(* IEC 61131-3 sources: RL_MAR/experiments/comparison/autoplc/results/deepseek-ai-DeepSeek-V3.2_20260508_111905/hard_92, 1 file *)

(* ---- hard_92_1.st ---- *)
FUNCTION_BLOCK FB_BreakerControlSystem
VAR_INPUT
    B10_1_Trip : BOOL;
    B10_1_Close : BOOL;
    B10_2_Trip : BOOL;
    B10_2_Close : BOOL;
    B10_12_Trip : BOOL;
    B10_12_Close : BOOL;
    B54_Trip : BOOL;
    B54_Close : BOOL;
    B55_Trip : BOOL;
    B55_Close : BOOL;
    B56_Trip : BOOL;
    B56_Close : BOOL;
    B57_Trip : BOOL;
    B57_Close : BOOL;
END_VAR
VAR_OUTPUT
    Point_1a : INT;
    Point_2a : INT;
    Point_3a : INT;
    Point_4a : INT;
    B10_1_Opened : BOOL;
    B10_1_Closed : BOOL;
    B10_2_Opened : BOOL;
    B10_2_Closed : BOOL;
    B10_12_Opened : BOOL;
    B10_12_Closed : BOOL;
    B54_Opened : BOOL;
    B54_Closed : BOOL;
    B55_Opened : BOOL;
    B55_Closed : BOOL;
    B56_Opened : BOOL;
    B56_Closed : BOOL;
    B57_Opened : BOOL;
    B57_Closed : BOOL;
END_VAR
VAR
    SEL86_OUT : INT;
    MOVE89_OUT : INT;
    SEL66_OUT : INT;
    MOVE69_OUT : INT;
    SEL96_OUT : INT;
    MOVE99_OUT : INT;
    SEL106_OUT : INT;
    MOVE109_OUT : INT;
END_VAR

VAR
    // Internal variables for state management
    bCondition1 : BOOL;
    bCondition2 : BOOL;
    bCondition3 : BOOL;
    bCondition4 : BOOL;
END_VAR

// Breaker B10_1 state management
IF B10_1_Close THEN
    B10_1_Closed := TRUE;
    B10_1_Opened := FALSE;
ELSIF B10_1_Trip THEN
    B10_1_Closed := FALSE;
    B10_1_Opened := TRUE;
END_IF;

// Breaker B10_2 state management
IF B10_2_Close THEN
    B10_2_Closed := TRUE;
    B10_2_Opened := FALSE;
ELSIF B10_2_Trip THEN
    B10_2_Closed := FALSE;
    B10_2_Opened := TRUE;
END_IF;

// Breaker B10_12 state management
IF B10_12_Close THEN
    B10_12_Closed := TRUE;
    B10_12_Opened := FALSE;
ELSIF B10_12_Trip THEN
    B10_12_Closed := FALSE;
    B10_12_Opened := TRUE;
END_IF;

// Breaker B54 state management
IF B54_Close THEN
    B54_Closed := TRUE;
    B54_Opened := FALSE;
ELSIF B54_Trip THEN
    B54_Closed := FALSE;
    B54_Opened := TRUE;
END_IF;

// Breaker B55 state management
IF B55_Close THEN
    B55_Closed := TRUE;
    B55_Opened := FALSE;
ELSIF B55_Trip THEN
    B55_Closed := FALSE;
    B55_Opened := TRUE;
END_IF;

// Breaker B56 state management
IF B56_Close THEN
    B56_Closed := TRUE;
    B56_Opened := FALSE;
ELSIF B56_Trip THEN
    B56_Closed := FALSE;
    B56_Opened := TRUE;
END_IF;

// Breaker B57 state management
IF B57_Close THEN
    B57_Closed := TRUE;
    B57_Opened := FALSE;
ELSIF B57_Trip THEN
    B57_Closed := FALSE;
    B57_Opened := TRUE;
END_IF;

// Calculate conditions for point outputs
bCondition1 := B54_Closed AND ((B10_12_Closed AND B10_1_Closed) OR B10_2_Closed);
bCondition2 := B55_Closed AND ((B10_12_Closed AND B10_1_Closed) OR B10_2_Closed);
bCondition3 := B56_Closed AND ((B10_12_Closed AND B10_2_Closed) OR B10_1_Closed);
bCondition4 := B57_Closed AND ((B10_12_Closed AND B10_2_Closed) OR B10_1_Closed);

// Calculate Point_1a
IF bCondition1 THEN
    Point_1a := 0;
ELSE
    Point_1a := 138;
END_IF;

// Calculate Point_2a
IF bCondition2 THEN
    Point_2a := 0;
ELSE
    Point_2a := 138;
END_IF;

// Calculate Point_3a
IF bCondition3 THEN
    Point_3a := 0;
ELSE
    Point_3a := 138;
END_IF;

// Calculate Point_4a
IF bCondition4 THEN
    Point_4a := 0;
ELSE
    Point_4a := 138;
END_IF;

// Internal variables (SELxx_OUT and MOVExx_OUT) are not used in the main logic
// but are kept as declared in the VAR section
SEL86_OUT := 0;
MOVE89_OUT := 0;
SEL66_OUT := 0;
MOVE69_OUT := 0;
SEL96_OUT := 0;
MOVE99_OUT := 0;
SEL106_OUT := 0;
MOVE109_OUT := 0;

END_FUNCTION_BLOCK
